{attribute 'no_explicit_call' := 'This FB is a CLASS and must be accessed using methods or properties'}
{attribute 'enable_dynamic_creation'}
FUNCTION_BLOCK ListForwardEnumerator EXTENDS Disposable IMPLEMENTS I_ForwardEnumerator, I_EventHandler
VAR
	parent : I_List;
	currentIndex : DINT := 0;
	invalid : BOOL := FALSE;
	moveNextCalled : BOOL := FALSE;
END_VAR

METHOD FB_exit : BOOL
VAR_INPUT
	bInCopyCode : BOOL; // if TRUE, the exit method is called for exiting an instance that is copied afterwards (online change).
END_VAR
IF bInCopyCode THEN
	RETURN;
END_IF

IF parent = 0 THEN
	RETURN;
END_IF

parent.OffEvent('OnChanged',THIS^);
parent.OffEvent('OnDisposed',THIS^);
END_METHOD

METHOD FB_init : BOOL
VAR_INPUT
	bInitRetains : BOOL; // if TRUE, the retain variables are initialized (warm start / cold start)
	bInCopyCode : BOOL;  // if TRUE, the instance afterwards gets moved into the copy code (online change)
	Parent : I_List;
END_VAR
Parent.OnEvent('OnChanged',THIS^);
Parent.OnEvent('OnDisposed',THIS^);
this^.parent := Parent;
END_METHOD

METHOD PUBLIC HandleEvent
VAR_INPUT
	Event : I_Event;
END_VAR
VAR
	changedEvent : I_CollectionChangedEvent;
	disposedEvent : I_CollectionDisposedEvent;
END_VAR
IF __QUERYINTERFACE(Event, changedEvent) THEN
	invalid := TRUE;
	currentIndex := 0;
ELSIF __QUERYINTERFACE(Event, disposedEvent) THEN
	parent := 0;
END_IF
END_METHOD

PROPERTY PUBLIC IsValid : BOOL
GET
IsValid := (NOT invalid AND parent <> 0);
END_GET
END_PROPERTY

METHOD MoveNext : BOOL
IF invalid THEN
    RETURN;
END_IF

IF parent = 0 THEN
    RETURN;
END_IF

IF parent.Count = 0 THEN
    RETURN;
END_IF

IF NOT moveNextCalled THEN
	MoveNext := moveNextCalled := TRUE;
	RETURN;
END_IF

IF currentIndex < parent.Count - 1 THEN
    currentIndex := currentIndex + 1;
    MoveNext := TRUE;
END_IF
END_METHOD

METHOD Reset
VAR_INPUT
END_VAR
moveNextCalled := FALSE;
currentIndex := 0;
END_METHOD

METHOD PUBLIC TryGet : BOOL
VAR_INPUT
	Destination : ANY;
END_VAR
IF invalid THEN
	RETURN;
END_IF

IF parent = 0 THEN
	RETURN;
END_IF

IF NOT moveNextCalled THEN
	RETURN;
END_IF

TryGet := parent.TryGetByIndex(currentIndex, Destination);
END_METHOD

METHOD TryGetTo : BOOL
VAR_INPUT
	DestinationAddress : PVOID;
	DestinationSize : UDINT;
END_VAR
IF invalid THEN
	RETURN;
END_IF

IF parent = 0 THEN
	RETURN;
END_IF

IF NOT moveNextCalled THEN
	RETURN;
END_IF

TryGetTo := parent.TryGetToByIndex(currentIndex, DestinationAddress, DestinationSize);
END_METHOD

END_FUNCTION_BLOCK

(* stored: Version 1.1.0.1, ProductVersion 3.1.4024.12
   POU ListForwardEnumerator: Id {71cbcc34-b058-4022-8d0f-92c2cf91e030}, SpecialFunc None
   Folder Constructor: Id {cdeb2947-3a90-4b8f-a836-b2e28e3f7057}
   Folder Destructor: Id {0508b0ce-2c85-4f37-8751-719fea7d3821}
   Method FB_exit: Id {a884428f-80e3-4ea4-ac89-94b01a155b6e}
   Method FB_init: Id {561615b3-2102-4e89-85a3-3eb981a30740}
   Method HandleEvent: Id {d7956ff3-1f96-468a-a2cd-01e1f741b627}
   Property IsValid: Id {0eb1db84-cd2b-4f80-9b94-dc9f9847529f}
   Get Get: Id {7fc3be42-663f-4bd2-bee5-b34cca659a44}
   Method MoveNext: Id {124806d4-b465-483c-825d-a72774a6ff60}
   Method Reset: Id {a8a10cb7-9f41-48bf-8314-7d421717f7a9}
   Method TryGet: Id {fc9b3816-84f5-4733-83b3-f353243e6fb9}
   Method TryGetTo: Id {c779c4e7-cbea-4286-b465-4d39f43aee99} *)
